Fanuc KAREL source: kt00029.KL

-- PROVISIONAL review KL for V1013-1; original PC SHA256 27f3a9c623240987926e882b2bc1e6db6363c098bb9cd5802a745cb7cd3a2b69
-- Incomplete behavior may be omitted. Consult companion uncertainty JSON. Do not deploy.
PROGRAM KT00029
%NOLOCKGROUP
VAR
  OUT : INTEGER
-- UNRESOLVED_DECL H1 type=002017
-- UNRESOLVED_DECL Y2 type=002018
BEGIN
  -- UNRESOLVED_PC offsets 5-19; opcodes 2E,22,9D,33,B4
  -- UNRESOLVED_PC offsets 24-38; opcodes 2E,22,9D,33,B2
  -- UNRESOLVED_PC offsets 43-68; opcodes 22,9D,33,B3,22,9D,33,B1,52,23
  -- UNRESOLVED_PC offsets 73-77; opcodes 7F
END KT00029
